// TIA Portal V17 export
TagTable "Codex_VBS_Loop_Tags"
  Codex_VBS_Input : WString  (1 s)
  Codex_VBS_Output : WString  (1 s)
